{attribute 'GeneratedUsingTerminal: EK1960-0000-0021'}
{attribute addProperty BoxType "EK1960-0000-0021"}
{attribute addProperty Id "Module_1_FSoEModule_1_FSoE_042BAFD398Module_2_FSOUTModule_2_FSOUT_8B7AA8A224Module_3_FSLOGICModule_3_FSLOGIC_DEAB45222WcStateAT %I*WcState_B516A2644InfoDataAT %I*InfoData_94A18F5E2"}
{attribute addProperty CRC "753075369"}
{attribute addProperty Size "130"}
TYPE EK1960_2CE304A9 EXTENDS EtcSlaveTerminalBase_947E5A46 :
STRUCT
	{attribute addProperty Name "Module_1_FSoE"}
	Module_1_FSoE : Module_1_FSoE_042BAFD3;
	{attribute addProperty Name "Module_2_FSOUT"}
	Module_2_FSOUT : Module_2_FSOUT_8B7AA8A2;
	{attribute addProperty Name "Module_3_FSLOGIC"}
	Module_3_FSLOGIC : Module_3_FSLOGIC_DEAB4522;
	{attribute addProperty Name "WcState"}
	WcState : WcState_B516A264;
	{attribute addProperty Name "InfoData"}
	InfoData : InfoData_94A18F5E;
END_STRUCT
END_TYPE

(* stored: Version 1.2.0.0, ProductVersion 3.1.4024.9
   DUT EK1960_2CE304A9: Id {36959502-b7b7-445c-908c-935c919a7228} *)
